(* CoDeSys 2.3 export: CreatePingReqMessage.EXP *)

(* POU MQTT-Utils/CreatePingReqMessage, ST *)
FUNCTION CreatePingReqMessage : UINT
VAR_INPUT
	pMessage		: POINTER TO BYTE;
END_VAR
VAR
	pDst			: POINTER TO BYTE;
	pSrc			: POINTER TO BYTE;
	clientIdLength	: BYTE;
END_VAR
(* Fixed header, byte 1, Control Packet type *)
pMessage^ := MQTT_MESSAGE_TYPE_PINGREQ;

(* Fixed header, byte 2, Remaining Length *)
pMessage := pMessage + 1;
pMessage^ := 0;

(* Return the total message length *)
CreatePingReqMessage := 2;
END_FUNCTION
